// Mitsubishi GX Works2 project: Exercicio time p on e of   PLC: Q03UDV

// task Task_01 (event TRUE, interval 0, priority 31): POU_01

PROGRAM POU_01
VAR
  TimerON : TON;
  TimerPonto : TP;
  TiOFF : TIME;
  TimerOF : TOF;
  TiON : TIME;
  TiPonto : TIME;
  Entrada : BOOL;
  Contador : CTD;
  VRA : BOOL;
  AMA : BOOL;
  VDA : BOOL;
END_VAR
(* structured ladder/FBD written out as ST: instructions are called as NAME(EN, inputs, outputs); _pN, _eN, _tN stand for wires *)
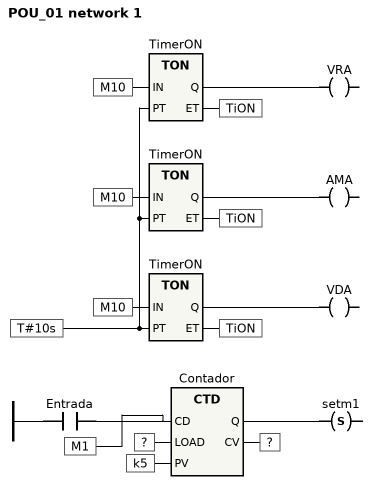
(* network 1 *)
TimerON(IN := M10, PT := T#10s, ET => TiON);
VRA := TimerON.Q;
TimerON(IN := M10, PT := T#10s, ET => TiON);
AMA := TimerON.Q;
TimerON(IN := M10, PT := T#10s, ET => TiON);
VDA := TimerON.Q;
Contador(CD := Entrada OR M1, LOAD := ?, PV := k5, CV => ?);
SET(Contador.Q, setm1);
END_PROGRAM
